FUNCTION_BLOCK FB_SimulatedIO
VAR_OUTPUT
	bRelayOn : BOOL := FALSE;
END_VAR
VAR CONSTANT
	PUMP_GAIN : REAL := 0.01;
	PASSIVE_LOSS : REAL := 0.001;
END_VAR

IF GVL_VAR.bPump THEN
	GVL_VAR.nPressure := GVL_VAR.nPressure + PUMP_GAIN;
ELSIF GVL_VAR.nPressure > 1 THEN
	GVL_VAR.nPressure := GVL_VAR.nPressure - PASSIVE_LOSS;
END_IF

END_FUNCTION_BLOCK

(* stored: Version 1.1.0.1, ProductVersion 3.1.4024.12
   POU FB_SimulatedIO: Id {0dda3bf4-0ef3-4e58-b3bf-1d433ae1dc6e}, SpecialFunc None *)
